TYPE ST_DOSOutputsMX :
STRUCT
	bOutputCh1	AT%Q*: BOOL;
	bOutputCh2	AT%Q*: BOOL;
	bOutputCh3	AT%Q*: BOOL;
	bOutputCh4	AT%Q*: BOOL;
	bOutputCh5	AT%Q*: BOOL;
	bOutputCh6	AT%Q*: BOOL;
	bOutputCh7	AT%Q*: BOOL;
	bOutputCh8	AT%Q*: BOOL;
END_STRUCT
END_TYPE

(* stored: Version 1.1.0.1
   DUT ST_DOSOutputsMX: Id {1520e8ca-b868-4e96-a953-15c66bdc4481} *)
